(* PLC project M3_18, Desconocido M3_18 1 *)
(* stored: creationDateTime 2025-05-15T11:40:54, modificationDateTime 2025-06-17T14:39:10 *)

PROGRAM Main
  VAR
    TON0 : TON;
    TON1 : TON;
    xPulso : BOOL;
    xActivar : BOOL;
    xM1 : BOOL;
    iMinutos : INT;
    CTU0 : CTU;
  END_VAR
  VAR  (* added by the conversion: wires and edge detectors of the diagram *)
    R_TRIG1 : R_TRIG;
  END_VAR

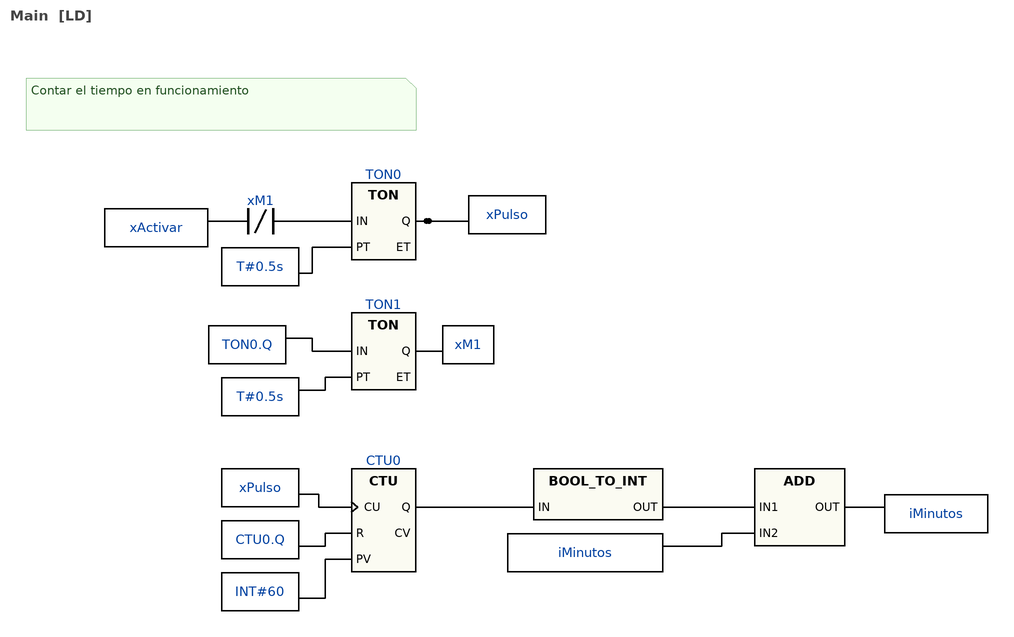
(* LD diagram, written out as Structured Text *)
(* Contar el tiempo en funcionamiento *)
TON0(IN := xActivar AND NOT xM1, PT := T#0.5s);
xPulso := TON0.Q;
TON1(IN := TON0.Q, PT := T#0.5s);
xM1 := TON1.Q;
R_TRIG1(CLK := xPulso);
CTU0(CU := R_TRIG1.Q, R := CTU0.Q, PV := INT#60);
iMinutos := BOOL_TO_INT(CTU0.Q) + iMinutos;
END_PROGRAM

CONFIGURATION Config0
  RESOURCE Res0 ON PLC
    TASK task0(INTERVAL := T#20ms, PRIORITY := 0);
    PROGRAM instance0 WITH task0 : Main;
  END_RESOURCE
END_CONFIGURATION
